//==================================================================================================
//							Beckhoff Automation Poland
//									18.04.2018
//	Struktura zawierajaca I/O odpowiedniego bloku
//  v1.0	|| TC v 3.1.4022.16		|| - pierwsza wersja
//==================================================================================================
TYPE ST_FBReadChannelErrorCodeIO:
STRUCT
	bExecute						: BOOL;								// Rising edge executes cmd
	bBusy							: BOOL;
	bError							: BOOL; 							// General error: parameter or CoE read.
	uiAdsErrId						: UINT;								// Forwarded output FB_CoERead_ByDriveRef
	uiSecErrId						: UINT;								// Sercos Error ID for AX5000, CanOpen error ID for AX8000
	uiChannelErrorCode				: UINT;								// 603F Error code	0x603F (Ch A)/ 0x683F (Ch B) 	UINT16
	{attribute 'displaymode':='hex'}
	uiChannelErrorCodeHex			: UINT;								// 603F Error code	0x603F (Ch A)/ 0x683F (Ch B) 	UINT16
END_STRUCT
END_TYPE

(* stored: Version 1.1.0.1, ProductVersion 3.1.4026.13, FileIdentifier ee770c7d6acac8b2f973e569679eaf3e3b17dc81, FileSignature 823769fd72a2274b98d4843c07a3aba2892c49cfa4cab8a049a0478c624e7a907b734e2904dad0e1259057056d2084603af6315e9fc72b668b710fca89aafdbf1eaa67e690d36cbee84a3104aeb0069ac34155d65b9b68303a58150c16c0e104bf0e29a1ec66f78d50433f6bc105e24c7063152b84fd1e35ecee821e0ea5ed95d6a78f2d50cbb4a56b90fd4ff57b8cc1851963e5159507ca593ff4ab9620868e42262dbafb84e554b38f09eaa6f81458152db4b4827ed31d638fbfac8dc3e2b7c6c2ff79424cf81f2268ac57c6c4623932ba2128cbeddf94707481e1353907b65bfd646239f34419798fe37be3e71c2b2e14a8f12cf959487feb8cd7d5c8308b
   DUT ST_FBReadChannelErrorCodeIO: Id {9d794b31-a9da-4fea-8a72-f3f3162fca6e} *)
